	                    #sFB_MCOConveyLinxAixController210(iUDT_AixConfig := #iUDT_Configuration."210".MCO_M01,
	                                                       iv_AixInputsModule := #iUDT_MotorInput210,
	                                                       ix_24vOk := #ix_24vOk,
	                                                       ix_SimulationModeActive := "DB_Memory".Simulation,
	                                                       ii_MotorPositionId := 1,
	                                                       qUDT_HMIStatus => #iqUDT_WorkstationStatus."210".MCO_M01,
	                                                       iqv_AixOutputsModule := #iqUDT_MotorOutput210,
	                                                       iqUDT_ConveyorInterface := #sUDT_Interface210,
	                                                       iqUDT_MCOStatistics := #iqUDT_WorkstationStatistics."210".MCO_M01);
	                END_REGION
	            END_REGION

	            REGION 211

	                REGION Displacement

	                    #sFB_Displacement211(#sUDT_Interface211);

	                END_REGION

	                REGION RAT

	                    IF #iUDT_Configuration.GlobalConfig.StationVariant = 1 OR #iUDT_Configuration.GlobalConfig.StationVariant = 2 THEN
	                        #sUDT_Handshake211C := #sUDT_Handshake190;
	                    ELSIF #iUDT_Configuration.GlobalConfig.StationVariant = 3 THEN
	                        #sUDT_Handshake211D := #sUDT_Handshake590;
	                    END_IF;


	                    #sFB_RightAngledTransfer211(iUDT_Configuration := #iUDT_Configuration."211".RightAngledTransfer,
	                                                iUDT_LowerConveyorConfiguration := #iUDT_Configuration."210".Conveyor,
	                                                iUDT_UpperConveyorConfiguration := #iUDT_Configuration."211".Conveyor,
	                                                iUDT_PECConfiguration := #iUDT_Configuration."210".PEC_EoS,
	                                                ii_DestinationA := 0,
	                                                ii_DestinationB := 0,
	                                                ii_DestinationC := 2,
	                                                ii_DestinationD := 0,
	                                                ix_HardwareOk := #iUDT_HardwareOk."210",
	                                                ix_400vOk := #ix_400vOk,
	                                                ix_24vOk := #ix_24vOk,
	                                                ix_SafetyOk := #ix_SafetyOk,
	                                                ix_AirPressureOk := #ix_AirPressureOk,
	                                                ix_SectionIsDown := #ix_SectionIsDown211,
	                                                ix_SectionIsUp := #ix_SectionIsUp211,
	                                                ix_ConveyorAAuto := false,
	                                                ix_ConveyorBAuto := false,
	                                                ix_ConveyorCAuto := #iqUDT_WorkstationCommonStatus."190".AutoON,
	                                                ix_ConveyorDAuto := false,
	                                                ix_PEC := #iUDT_MotorInput210.AllSensorPortInputs.LeftSensor,
	                                                ix_ExternalReceiveRequestA := FALSE,
	                                                ix_ExternalReceiveRequestB := FALSE,
	                                                ix_ExternalReceiveRequestC := #sx_LeftPushOutActiveStation1,
	                                                ix_ExternalReceiveRequestD := FALSE,
	                                                ix_PECInfeedC := #iqUDT_WorkstationStatus."190".PEC_EoS.PEC,
	                                                qUDT_HMIRATStatus => #iqUDT_WorkstationStatus."211".RightAngledTransfer,
	                                                qUDT_HMIConveyorStatus => #iqUDT_WorkstationStatus."210".Conveyor,
	                                                qUDT_HMIPECStatus => #iqUDT_WorkstationStatus."210".PEC_EoS,
	                                                qUDT_RATStatus => #iqUDT_WorkstationCommonStatus."211",
	                                                qUDT_ConveyorStatus => #iqUDT_WorkstationCommonStatus."210",
	                                                qx_PopupControl => #qx_PopupControl211,
	                                                qx_ExternalSendRequestA => #tx_dummy,
	                                                qx_ExternalSendRequestB => #tx_dummy,
	                                                qx_ExternalSendRequestC => #tx_dummy,
	                                                qx_ExternalSendRequestD => #tx_dummy,
	                                                iqUDT_EquipmentControl := #iqUDT_EquipmentControl,
	                                                iqUDT_RATCommand := #iqUDT_WorkstationCommands."211".RightAngledTransfer,
	                                                iqUDT_ConveyorCommand := #iqUDT_WorkstationCommands."210".Conveyor,
	                                                iqUDT_RATStatistics := #iqUDT_WorkstationStatistics."211".RightAngledTransfer,
	                                                iqUDT_ConveyorStatistics := #iqUDT_WorkstationStatistics."210".Conveyor,
	                                                iqUDT_PECStatistics := #iqUDT_WorkstationStatistics."210".PEC_EoS,
	                                                iqUDT_HandShakeConveyorA := #tUDT_DummyConveyorHandshake,
	                                                iqUDT_HandShakeConveyorB := #sUDT_Handshake210,
	                                                iqUDT_HandShakeConveyorC := #sUDT_Handshake211C,
	                                                iqUDT_HandShakeConveyorD := #sUDT_Handshake211D,
	                                                iqUDT_LowerConveyorInterface := #sUDT_Interface210,
	                                                iqUDT_UpperConveyorInterface := #sUDT_Interface211,
	                                                iqUDT_RATPositioning := #iqUDT_RATPositioning210,
	                                                iqUDT_BladeStopEoSInterface := #tUDT_DummyBladeStop,
	                                                iqUDT_BladeStopBoSInterface := #tUDT_DummyBladeStop);

	                END_REGION

	                IF #iUDT_Configuration.GlobalConfig.StationVariant = 1 OR #iUDT_Configuration.GlobalConfig.StationVariant = 2 THEN
	                    #sUDT_Handshake190 := #sUDT_Handshake211C;
	                ELSIF #iUDT_Configuration.GlobalConfig.StationVariant = 3 THEN
	                    #sUDT_Handshake590 := #sUDT_Handshake211D;
	                END_IF;


	                REGION MCO

	                    #sFB_MCOConveyLinxAixController211(iUDT_AixConfig := #iUDT_Configuration."211".MCO_M01,
	                                                       iv_AixInputsModule := #iUDT_MotorInput210,
	                                                       ii_PositionSetpoint := #iqUDT_RATPositioning210.Upper.EndPosition,
	                                                       ix_24vOk := #ix_24vOk,
	                                                       ix_SimulationModeActive := "DB_Memory".Simulation,
	                                                       ii_MotorPositionId := 2,
	                                                       ix_StartPositioning := #iqUDT_RATPositioning210.Upper.Start,
	                                                       ix_ResetPosition := #iqUDT_RATPositioning210.Upper.ResetPosition,
	                                                       qUDT_HMIStatus => #iqUDT_WorkstationStatus."211".MCO_M01,
	                                                       qx_Positioned => #iqUDT_RATPositioning210.Upper.Done,
	                                                       iqv_AixOutputsModule := #iqUDT_MotorOutput210,
	                                                       iqUDT_ConveyorInterface := #sUDT_Interface211,
	                                                       iqUDT_MCOStatistics := #iqUDT_WorkstationStatistics."211".MCO_M01);
	                END_REGION

	            END_REGION

	            REGION 220

	                REGION Displacement

	                    #sFB_Displacement220(#sUDT_Interface220);

	                END_REGION

	                REGION MCO

	                    #sFB_MCOConveyLinxAixController220(iUDT_AixConfig := #iUDT_Configuration."220".MCO_M01,
	                                                       iv_AixInputsModule := #iUDT_MotorInput220,
	                                                       ii_PositionSetpoint := #iqUDT_RATPositioning220.Lower.EndPosition,
	                                                       ix_24vOk := #ix_24vOk,
	                                                       ix_SimulationModeActive := "DB_Memory".Simulation,
	                                                       ii_MotorPositionId := 1,
	                                                       ix_StartPositioning := #iqUDT_RATPositioning220.Lower.Start,
	                                                       ix_ResetPosition := #iqUDT_RATPositioning220.Lower.ResetPosition,
	                                                       qUDT_HMIStatus => #iqUDT_WorkstationStatus."220".MCO_M01,
	                                                       qx_Positioned => #iqUDT_RATPositioning220.Lower.Done,
	                                                       iqv_AixOutputsModule := #iqUDT_MotorOutput220,
	                                                       iqUDT_ConveyorInterface := #sUDT_Interface220,
	                                                       iqUDT_MCOStatistics := #iqUDT_WorkstationStatistics."220".MCO_M01);
	                END_REGION
	            END_REGION

	            REGION 221

	                REGION Displacement

	                    #sFB_Displacement221(#sUDT_Interface221);

	                END_REGION

	                REGION RAT

	                    IF #iUDT_Configuration.GlobalConfig.StationVariant = 1 OR #iUDT_Configuration.GlobalConfig.StationVariant = 2 THEN
	                        #sUDT_Handshake221C := #sUDT_Handshake350;
	                    ELSIF #iUDT_Configuration.GlobalConfig.StationVariant = 3 THEN
	                        #sUDT_Handshake221D := #sUDT_Handshake750;
	                    END_IF;


	                    #sFB_RightAngledTransfer221(iUDT_Configuration := #iUDT_Configuration."221".RightAngledTransfer,
	                                                iUDT_LowerConveyorConfiguration := #iUDT_Configuration."220".Conveyor,
	                                                iUDT_UpperConveyorConfiguration := #iUDT_Configuration."221".Conveyor,
	                                                iUDT_PECConfiguration := #iUDT_Configuration."220".PEC_EoS,
	                                                ii_DestinationA := 2,
	                                                ii_DestinationB := 0,
	                                                ii_DestinationC := 2,
	                                                ii_DestinationD := 0,
	                                                ix_HardwareOk := #iUDT_HardwareOk."220",
	                                                ix_400vOk := #ix_400vOk,
	                                                ix_24vOk := #ix_24vOk,
	                                                ix_SafetyOk := #ix_SafetyOk,
	                                                ix_AirPressureOk := #ix_AirPressureOk,
	                                                ix_SectionIsDown := #ix_SectionIsDown221,
	                                                ix_SectionIsUp := #ix_SectionIsUp221,
	                                                ix_ConveyorAAuto := #iqUDT_WorkstationCommonStatus."210".AutoON,
	                                                ix_ConveyorBAuto := false,
	                                                ix_ConveyorCAuto := #iqUDT_WorkstationCommonStatus."350".AutoON,
	                                                ix_ConveyorDAuto := false,
	                                                ix_PEC := #iUDT_MotorInput220.AllSensorPortInputs.LeftSensor,
	                                                ix_ExternalReceiveRequestA := NOT #iqUDT_WorkstationStatus."210".PEC_EoS.PEC,
	                                                ix_ExternalReceiveRequestB := FALSE,
	                                                ix_ExternalReceiveRequestC := NOT #iqUDT_WorkstationStatus."350".PEC_EoS.PEC,
	                                                ix_ExternalReceiveRequestD := TRUE,
	                                                ix_PECInfeedA := #iqUDT_WorkstationStatus."210".PEC_EoS.PEC,
	                                                ix_PECInfeedC := #iqUDT_WorkstationStatus."350".PEC_EoS.PEC,
	                                                qUDT_HMIRATStatus => #iqUDT_WorkstationStatus."221".RightAngledTransfer,
	                                                qUDT_HMIConveyorStatus => #iqUDT_WorkstationStatus."220".Conveyor,
	                                                qUDT_HMIPECStatus => #iqUDT_WorkstationStatus."220".PEC_EoS,
	                                                qUDT_RATStatus => #iqUDT_WorkstationCommonStatus."221",
	                                                qUDT_ConveyorStatus => #iqUDT_WorkstationCommonStatus."220",
	                                                qx_PopupControl => #qx_PopupControl221,
	                                                qx_ExternalSendRequestA => #tx_dummy,
	                                                qx_ExternalSendRequestB => #tx_dummy,
	                                                qx_ExternalSendRequestC => #tx_dummy,
	                                                qx_ExternalSendRequestD => #tx_dummy,
	                                                iqUDT_EquipmentControl := #iqUDT_EquipmentControl,
	                                                iqUDT_RATCommand := #iqUDT_WorkstationCommands."221".RightAngledTransfer,
	                                                iqUDT_ConveyorCommand := #iqUDT_WorkstationCommands."220".Conveyor,
	                                                iqUDT_RATStatistics := #iqUDT_WorkstationStatistics."221".RightAngledTransfer,
	                                                iqUDT_ConveyorStatistics := #iqUDT_WorkstationStatistics."220".Conveyor,
	                                                iqUDT_PECStatistics := #iqUDT_WorkstationStatistics."220".PEC_EoS,
	                                                iqUDT_HandShakeConveyorA := #sUDT_Handshake210,
	                                                iqUDT_HandShakeConveyorB := #iqUDT_HandshakeDownstream220,
	                                                iqUDT_HandShakeConveyorC := #sUDT_Handshake221C,
	                                                iqUDT_HandShakeConveyorD := #sUDT_Handshake221D,
	                                                iqUDT_LowerConveyorInterface := #sUDT_Interface220,
	                                                iqUDT_UpperConveyorInterface := #sUDT_Interface221,
	                                                iqUDT_RATPositioning := #iqUDT_RATPositioning220,
	                                                iqUDT_BladeStopEoSInterface := #tUDT_DummyBladeStop,
	                                                iqUDT_BladeStopBoSInterface := #tUDT_DummyBladeStop);

	                END_REGION

	                IF #iUDT_Configuration.GlobalConfig.StationVariant = 1 OR #iUDT_Configuration.GlobalConfig.StationVariant = 2 THEN
	                    #sUDT_Handshake350 := #sUDT_Handshake221C;
	                ELSIF #iUDT_Configuration.GlobalConfig.StationVariant = 3 THEN
	                    #sUDT_Handshake750 := #sUDT_Handshake221D;
	                END_IF;

	                REGION MCO

	                    #sFB_MCOConveyLinxAixController221(iUDT_AixConfig := #iUDT_Configuration."221".MCO_M01,
	                                                       iv_AixInputsModule := #iUDT_MotorInput220,
	                                                       ii_PositionSetpoint := #iqUDT_RATPositioning220.Upper.EndPosition,
	                                                       ix_24vOk := #ix_24vOk,
	                                                       ix_SimulationModeActive := "DB_Memory".Simulation,
	                                                       ii_MotorPositionId := 2,
	                                                       ix_StartPositioning := #iqUDT_RATPositioning220.Upper.Start,
	                                                       ix_ResetPosition := #iqUDT_RATPositioning220.Upper.ResetPosition,
	                                                       qUDT_HMIStatus => #iqUDT_WorkstationStatus."221".MCO_M01,
	                                                       qx_Positioned => #iqUDT_RATPositioning220.Upper.Done,
	                                                       iqv_AixOutputsModule := #iqUDT_MotorOutput220,
	                                                       iqUDT_ConveyorInterface := #sUDT_Interface221,
	                                                       iqUDT_MCOStatistics := #iqUDT_WorkstationStatistics."221".MCO_M01);
	                END_REGION
	            END_REGION

	            REGION 310

	                REGION Displacement

	                    #sFB_Displacement310(#sUDT_Interface310);

	                END_REGION

	                REGION EOS
	                    #sFB_PEC310(ix_PEC := NOT #iUDT_MotorInput310.AllSensorPortInputs.LeftSensor,
	                                iUDT_PECConfiguration := #iUDT_Configuration."310".PEC_Eos,
	                                qx_PECFiltered => #tx_dummy,
	                                qUDT_HMIStatus => #iqUDT_WorkstationStatus."310".PEC_EoS,
	                                iqUDT_ConveyorInterface := #sUDT_Interface310,
	                                iqUDT_PECStatistics := #iqUDT_WorkstationStatistics."310".PEC_EoS);

	                END_REGION

	                REGION Conveyor

	                    #sFB_Conveyor310(iUDT_ConveyorConfiguration := #iUDT_Configuration."310".Conveyor,
	                                     idi_PECEoSDistance := #iUDT_Configuration."310".PEC_Eos.Distance,
	                                     idi_PECBoSDistance := 0,
	                                     ii_ExternalSpeed := 0,
	                                     ix_SafetyOk := #ix_SafetyOk,
	                                     ix_24vOk := #ix_24vOk,
	                                     ix_400vOk := #ix_400vOk,
	                                     ix_HardwareOk := #iUDT_HardwareOk."310",
	                                     ix_PECEoS := #iqUDT_WorkstationStatus."310".PEC_EoS.PEC,
	                                     ix_PECBoS := TRUE,
	                                     ix_ReverseDirection := FALSE,
	                                     ix_ExternalRequestDieBack := FALSE,
	                                     ix_ExternalRequestHold := #sx_LeftExternalRequestHold310,
	                                     ix_ResetEnergySave := FALSE,
	                                     qUDT_HMIStatus => #iqUDT_WorkstationStatus."310".Conveyor,
	                                     qUDT_Status => #iqUDT_WorkstationCommonStatus."310",
	                                     iqUDT_EquipmentControl := #iqUDT_EquipmentControl,
	                                     iqUDT_ConveyorCommand := #iqUDT_WorkstationCommands."310".Conveyor,
	                                     iqUDT_ConveyorInterface := #sUDT_Interface310,
	                                     iqUDT_HandShakeUp := #tUDT_DummyConveyorHandshake,
	                                     iqUDT_HandShake := #sUDT_Handshake310,
	                                     iqUDT_Statistics := #iqUDT_WorkstationStatistics."310".Conveyor);
	                END_REGION

	                REGION MCO

	                    #sFB_MCOConveyLinxAixController310(iUDT_AixConfig := #iUDT_Configuration."310".MCO_M01,
	                                                       iv_AixInputsModule := #iUDT_MotorInput310,
	                                                       ix_24vOk := #ix_24vOk,
	                                                       ix_SimulationModeActive := "DB_Memory".Simulation,
	                                                       ii_MotorPositionId := 1,
	                                                       qUDT_HMIStatus => #iqUDT_WorkstationStatus."310".MCO_M01,
	                                                       iqv_AixOutputsModule := #iqUDT_MotorOutput310,
	                                                       iqUDT_ConveyorInterface := #sUDT_Interface310,
	                                                       iqUDT_MCOStatistics := #iqUDT_WorkstationStatistics."310".MCO_M01);
	                END_REGION

	            END_REGION

	            REGION 320

	                REGION Displacement

	                    #sFB_Displacement320(#sUDT_Interface320);

	                END_REGION

	                REGION EOS
	                    #sFB_PEC320(ix_PEC := NOT #iUDT_MotorInput310.AllSensorPortInputs.RightSensor,
	                                iUDT_PECConfiguration := #iUDT_Configuration."320".PEC_Eos,
	                                qx_PECFiltered => #tx_dummy,
	                                qUDT_HMIStatus => #iqUDT_WorkstationStatus."320".PEC_EoS,
	                                iqUDT_ConveyorInterface := #sUDT_Interface320,
	                                iqUDT_PECStatistics := #iqUDT_WorkstationStatistics."320".PEC_EoS);


	                END_REGION

	                REGION Conveyor

	                    #sFB_Conveyor320(iUDT_ConveyorConfiguration := #iUDT_Configuration."320".Conveyor,
	                                     idi_PECEoSDistance := #iUDT_Configuration."320".PEC_Eos.Distance,
	                                     idi_PECBoSDistance := 0,
	                                     ii_ExternalSpeed := 0,
	                                     ix_SafetyOk := #ix_SafetyOk,
	                                     ix_24vOk := #ix_24vOk,
	                                     ix_400vOk := #ix_400vOk,
	                                     ix_HardwareOk := #iUDT_HardwareOk."320",
	                                     ix_PECEoS := #iqUDT_WorkstationStatus."320".PEC_EoS.PEC,
	                                     ix_PECBoS := TRUE,
	                                     ix_ReverseDirection := FALSE,
	                                     ix_ExternalRequestDieBack := FALSE,
	                                     ix_ExternalRequestHold := #sx_LeftExternalRequestHold320,
	                                     ix_ResetEnergySave := FALSE,
	                                     qUDT_HMIStatus => #iqUDT_WorkstationStatus."320".Conveyor,
	                                     qUDT_Status => #iqUDT_WorkstationCommonStatus."320",
	                                     iqUDT_EquipmentControl := #iqUDT_EquipmentControl,
	                                     iqUDT_ConveyorCommand := #iqUDT_WorkstationCommands."320".Conveyor,
	                                     iqUDT_ConveyorInterface := #sUDT_Interface320,
	                                     iqUDT_HandShakeUp := #sUDT_Handshake310,
	                                     iqUDT_HandShake := #sUDT_Handshake320,
	                                     iqUDT_Statistics := #iqUDT_WorkstationStatistics."320".Conveyor);
	                END_REGION

	                REGION MCO

	                    #sFB_MCOConveyLinxAixController320(iUDT_AixConfig := #iUDT_Configuration."320".MCO_M01,
	                                                       iv_AixInputsModule := #iUDT_MotorInput310,
	                                                       ix_24vOk := #ix_24vOk,
	                                                       ix_SimulationModeActive := "DB_Memory".Simulation,
	                                                       ii_MotorPositionId := 2,
	                                                       qUDT_HMIStatus => #iqUDT_WorkstationStatus."320".MCO_M01,
	                                                       iqv_AixOutputsModule := #iqUDT_MotorOutput310,
	                                                       iqUDT_ConveyorInterface := #sUDT_Interface320,
	                                                       iqUDT_MCOStatistics := #iqUDT_WorkstationStatistics."320".MCO_M01);
	                END_REGION

	            END_REGION

	            REGION 330

	                REGION Displacement

	                    #sFB_Displacement330(#sUDT_Interface330);

	                END_REGION

	                REGION EOS
	                    #sFB_PEC330(ix_PEC := NOT #iUDT_MotorInput330.AllSensorPortInputs.LeftSensor,
	                                iUDT_PECConfiguration := #iUDT_Configuration."330".PEC_Eos,
	                                qx_PECFiltered => #tx_dummy,
	                                qUDT_HMIStatus => #iqUDT_WorkstationStatus."330".PEC_EoS,
	                                iqUDT_ConveyorInterface := #sUDT_Interface330,
	                                iqUDT_PECStatistics := #iqUDT_WorkstationStatistics."330".PEC_EoS);


	                END_REGION

	                REGION Conveyor

	                    #sFB_Conveyor330(iUDT_ConveyorConfiguration := #iUDT_Configuration."330".Conveyor,
	                                     idi_PECEoSDistance := #iUDT_Configuration."330".PEC_Eos.Distance,
	                                     idi_PECBoSDistance := 0,
	                                     ii_ExternalSpeed := 0,
	                                     ix_SafetyOk := #ix_SafetyOk,
	                                     ix_24vOk := #ix_24vOk,
	                                     ix_400vOk := #ix_400vOk,
	                                     ix_HardwareOk := #iUDT_HardwareOk."330",
	                                     ix_PECEoS := #iqUDT_WorkstationStatus."330".PEC_EoS.PEC,
	                                     ix_PECBoS := TRUE,
	                                     ix_ReverseDirection := FALSE,
	                                     ix_ExternalRequestDieBack := FALSE,
	                                     ix_ExternalRequestHold := #sx_LeftExternalRequestHold330,
	                                     ix_ResetEnergySave := FALSE,
	                                     qUDT_HMIStatus => #iqUDT_WorkstationStatus."330".Conveyor,
	                                     qUDT_Status => #iqUDT_WorkstationCommonStatus."330",
	                                     iqUDT_EquipmentControl := #iqUDT_EquipmentControl,
	                                     iqUDT_ConveyorCommand := #iqUDT_WorkstationCommands."330".Conveyor,
	                                     iqUDT_ConveyorInterface := #sUDT_Interface330,
	                                     iqUDT_HandShakeUp := #sUDT_Handshake320,
	                                     iqUDT_HandShake := #sUDT_Handshake330,
	                                     iqUDT_Statistics := #iqUDT_WorkstationStatistics."330".Conveyor);
	                END_REGION

	                REGION MCO

	                    #sFB_MCOConveyLinxAixController330(iUDT_AixConfig := #iUDT_Configuration."330".MCO_M01,
	                                                       iv_AixInputsModule := #iUDT_MotorInput330,
	                                                       ix_24vOk := #ix_24vOk,
	                                                       ix_SimulationModeActive := "DB_Memory".Simulation,
	                                                       ii_MotorPositionId := 1,
	                                                       qUDT_HMIStatus => #iqUDT_WorkstationStatus."330".MCO_M01,
	                                                       iqv_AixOutputsModule := #iqUDT_MotorOutput330,
	                                                       iqUDT_ConveyorInterface := #sUDT_Interface330,
	                                                       iqUDT_MCOStatistics := #iqUDT_WorkstationStatistics."330".MCO_M01);
	                END_REGION
	            END_REGION

	            REGION 340

	                REGION Displacement

	                    #sFB_Displacement340(#sUDT_Interface340);

	                END_REGION

	                REGION EOS
	                    #sFB_PEC340(ix_PEC := NOT #iUDT_MotorInput330.AllSensorPortInputs.RightSensor,
	                                iUDT_PECConfiguration := #iUDT_Configuration."340".PEC_Eos,
	                                qx_PECFiltered => #tx_dummy,
	                                qUDT_HMIStatus => #iqUDT_WorkstationStatus."340".PEC_EoS,
	                                iqUDT_ConveyorInterface := #sUDT_Interface340,
	                                iqUDT_PECStatistics := #iqUDT_WorkstationStatistics."340".PEC_EoS);


	                END_REGION


	                REGION Conveyor

	                    #sFB_Conveyor340(iUDT_ConveyorConfiguration := #iUDT_Configuration."340".Conveyor,
	                                     idi_PECEoSDistance := #iUDT_Configuration."340".PEC_Eos.Distance,
	                                     idi_PECBoSDistance := 0,
	                                     ii_ExternalSpeed := 0,
	                                     ix_SafetyOk := #ix_SafetyOk,
	                                     ix_24vOk := #ix_24vOk,
	                                     ix_400vOk := #ix_400vOk,
	                                     ix_HardwareOk := #iUDT_HardwareOk."340",
	                                     ix_PECEoS := #iqUDT_WorkstationStatus."340".PEC_EoS.PEC,
	                                     ix_PECBoS := TRUE,
	                                     ix_ReverseDirection := FALSE,
	                                     ix_ExternalRequestDieBack := FALSE,
	                                     ix_ExternalRequestHold := #sx_LeftExternalRequestHold340,
	                                     ix_ResetEnergySave := FALSE,
	                                     qUDT_HMIStatus => #iqUDT_WorkstationStatus."340".Conveyor,
	                                     qUDT_Status => #iqUDT_WorkstationCommonStatus."340",
	                                     iqUDT_EquipmentControl := #iqUDT_EquipmentControl,
	                                     iqUDT_ConveyorCommand := #iqUDT_WorkstationCommands."340".Conveyor,
	                                     iqUDT_ConveyorInterface := #sUDT_Interface340,
	                                     iqUDT_HandShakeUp := #sUDT_Handshake330,
	                                     iqUDT_HandShake := #sUDT_Handshake340,
	                                     iqUDT_Statistics := #iqUDT_WorkstationStatistics."340".Conveyor);
	                END_REGION

	                REGION MCO

	                    #sFB_MCOConveyLinxAixController340(iUDT_AixConfig := #iUDT_Configuration."340".MCO_M01,
	                                                       iv_AixInputsModule := #iUDT_MotorInput330,
	                                                       ix_24vOk := #ix_24vOk,
	                                                       ix_SimulationModeActive := "DB_Memory".Simulation,
	                                                       ii_MotorPositionId := 2,
	                                                       qUDT_HMIStatus => #iqUDT_WorkstationStatus."340".MCO_M01,
	                                                       iqv_AixOutputsModule := #iqUDT_MotorOutput330,
	                                                       iqUDT_ConveyorInterface := #sUDT_Interface340,
	                                                       iqUDT_MCOStatistics := #iqUDT_WorkstationStatistics."340".MCO_M01);
	                END_REGION
	            END_REGION

	            REGION 350

	                REGION Displacement

	                    #sFB_Displacement350(#sUDT_Interface350);

	                END_REGION

	                REGION EOS
	                    #sFB_PEC350(ix_PEC := NOT #iUDT_MotorInput350.AllSensorPortInputs.LeftSensor,
	                                iUDT_PECConfiguration := #iUDT_Configuration."350".PEC_Eos,
	                                qx_PECFiltered => #tx_dummy,
	                                qUDT_HMIStatus => #iqUDT_WorkstationStatus."350".PEC_EoS,
	                                iqUDT_ConveyorInterface := #sUDT_Interface350,
	                                iqUDT_PECStatistics := #iqUDT_WorkstationStatistics."350".PEC_EoS);

	                END_REGION

	                REGION Conveyor

	                    #sUDT_Handshake350.RTR := #sUDT_Handshake350.RTR OR #iqUDT_WorkstationStatus."350".PEC_EoS.PEC;

	                    #sFB_Conveyor350(iUDT_ConveyorConfiguration := #iUDT_Configuration."350".Conveyor,
	                                     idi_PECEoSDistance := #iUDT_Configuration."350".PEC_Eos.Distance,
	                                     idi_PECBoSDistance := 0,
	                                     ii_ExternalSpeed := 0,
	                                     ix_SafetyOk := #ix_SafetyOk,
	                                     ix_24vOk := #ix_24vOk,
	                                     ix_400vOk := #ix_400vOk,
	                                     ix_HardwareOk := #iUDT_HardwareOk."350",
	                                     ix_PECEoS := #iqUDT_WorkstationStatus."350".PEC_EoS.PEC,
	                                     ix_PECBoS := TRUE,
	                                     ix_ReverseDirection := FALSE,
	                                     ix_ExternalRequestDieBack := FALSE,
	                                     ix_ExternalRequestHold := #sx_LeftExternalRequestHold350,
	                                     ix_ResetEnergySave := FALSE,
	                                     qUDT_HMIStatus => #iqUDT_WorkstationStatus."350".Conveyor,
	                                     qUDT_Status => #iqUDT_WorkstationCommonStatus."350",
	                                     iqUDT_EquipmentControl := #iqUDT_EquipmentControl,
	                                     iqUDT_ConveyorCommand := #iqUDT_WorkstationCommands."350".Conveyor,
	                                     iqUDT_ConveyorInterface := #sUDT_Interface350,
	                                     iqUDT_HandShakeUp := #sUDT_Handshake340,
	                                     iqUDT_HandShake := #sUDT_Handshake350,
	                                     iqUDT_Statistics := #iqUDT_WorkstationStatistics."350".Conveyor);
	                END_REGION

	                REGION MCO

	                    #sFB_MCOConveyLinxAixController350(iUDT_AixConfig := #iUDT_Configuration."350".MCO_M01,
	                                                       iv_AixInputsModule := #iUDT_MotorInput350,
	                                                       ix_24vOk := #ix_24vOk,
	                                                       ix_SimulationModeActive := "DB_Memory".Simulation,
	                                                       ii_MotorPositionId := 1,
	                                                       qUDT_HMIStatus => #iqUDT_WorkstationStatus."350".MCO_M01,
	                                                       iqv_AixOutputsModule := #iqUDT_MotorOutput350,
	                                                       iqUDT_ConveyorInterface := #sUDT_Interface350,
	                                                       iqUDT_MCOStatistics := #iqUDT_WorkstationStatistics."350".MCO_M01);
	                END_REGION
	            END_REGION

	            REGION 360

	                REGION Displacement
	                    #sFB_Displacement360(#sUDT_Interface360);

	                END_REGION


	                REGION Conveyor

	                    #sUDT_Handshake360.RTR := TRUE;

	                    #sFB_Conveyor360(iUDT_ConveyorConfiguration := #iUDT_Configuration."360".Conveyor,
	                                     idi_PECEoSDistance := 0,
	                                     idi_PECBoSDistance := 0,
	                                     ii_ExternalSpeed := 0,
	                                     ix_SafetyOk := #ix_SafetyOk,
	                                     ix_24vOk := #ix_24vOk,
	                                     ix_400vOk := #ix_400vOk,
	                                     ix_HardwareOk := #iUDT_HardwareOk."360",
	                                     ix_PECEoS := TRUE,
	                                     ix_PECBoS := TRUE,
	                                     ix_ReverseDirection := false,
	                                     ix_ExternalRequestDieBack := false,
	                                     ix_ExternalRequestHold := #sx_Hold360,
	                                     ix_ResetEnergySave := false,
	                                     qUDT_HMIStatus => #iqUDT_WorkstationStatus."360".Conveyor,
	                                     qUDT_Status => #iqUDT_WorkstationCommonStatus."360",
	                                     iqUDT_EquipmentControl := #iqUDT_EquipmentControl,
	                                     iqUDT_ConveyorCommand := #iqUDT_WorkstationCommands."360".Conveyor,
	                                     iqUDT_ConveyorInterface := #sUDT_Interface360,
	                                     iqUDT_HandShakeUp := #sUDT_HandshakeUp360,
	                                     iqUDT_HandShake := #sUDT_Handshake360,
	                                     iqUDT_Statistics := #iqUDT_WorkstationStatistics."360".Conveyor);

	                END_REGION


	                REGION MCO
	                    #sFB_MCOConveyLinxAixController360(iUDT_AixConfig := #iUDT_Configuration."360".MCO_M01,
	                                                       iv_AixInputsModule := #iUDT_MotorInput360,
	                                                       ii_MotorPositionId := 1,
	                                                       ix_24vOk := #ix_24vOk,
	                                                       ix_SimulationModeActive := "DB_Memory".Simulation,
	                                                       qUDT_HMIStatus => #iqUDT_WorkstationStatus."360".MCO_M01,
	                                                       iqv_AixOutputsModule := #iqUDT_MotorOutput360,
	                                                       iqUDT_ConveyorInterface := #sUDT_Interface360,
	                                                       iqUDT_MCOStatistics := #iqUDT_WorkstationStatistics."360".MCO_M01);

	                END_REGION

	            END_REGION

	            REGION 370
	                REGION Displacement
	                    #sFB_Displacement370(#sUDT_Interface370);

	                END_REGION

	                REGION Conveyor

	                    #sUDT_Handshake370.RTR := TRUE;

	                    #sFB_Conveyor370(iUDT_ConveyorConfiguration := #iUDT_Configuration."370".Conveyor,
	                                     idi_PECEoSDistance := 0,
	                                     idi_PECBoSDistance := 0,
	                                     ii_ExternalSpeed := 0,
	                                     ix_SafetyOk := #ix_SafetyOk,
	                                     ix_24vOk := #ix_24vOk,
	                                     ix_400vOk := #ix_400vOk,
	                                     ix_HardwareOk := #iUDT_HardwareOk."360",
	                                     ix_PECEoS := TRUE,
	                                     ix_PECBoS := TRUE,
	                                     ix_ReverseDirection := false,
	                                     ix_ExternalRequestDieBack := false,
	                                     ix_ExternalRequestHold := #sx_Hold370,
	                                     ix_ResetEnergySave := false,
	                                     qUDT_HMIStatus => #iqUDT_WorkstationStatus."370".Conveyor,
	                                     qUDT_Status => #iqUDT_WorkstationCommonStatus."370",
	                                     iqUDT_EquipmentControl := #iqUDT_EquipmentControl,
	                                     iqUDT_ConveyorCommand := #iqUDT_WorkstationCommands."370".Conveyor,
	                                     iqUDT_ConveyorInterface := #sUDT_Interface370,
	                                     iqUDT_HandShakeUp := #sUDT_HandshakeUp370,
	                                     iqUDT_HandShake := #sUDT_Handshake370,
	                                     iqUDT_Statistics := #iqUDT_WorkstationStatistics."370".Conveyor);

	                END_REGION


	                REGION MCO
	                    #sFB_MCOConveyLinxAixController370(iUDT_AixConfig := #iUDT_Configuration."370".MCO_M01,
	                                                       iv_AixInputsModule := #iUDT_MotorInput360,
	                                                       ii_MotorPositionId := 2,
	                                                       ii_PositionSetpoint := 0,
	                                                       ix_24vOk := #ix_24vOk,
	                                                       ix_SimulationModeActive := "DB_Memory".Simulation,
	                                                       ix_StartPositioning := false,
	                                                       ix_ResetPosition := false,
	                                                       qUDT_HMIStatus => #iqUDT_WorkstationStatus."370".MCO_M01,
	                                                       iqv_AixOutputsModule := #iqUDT_MotorOutput360,
	                                                       iqUDT_ConveyorInterface := #sUDT_Interface370,
	                                                       iqUDT_MCOStatistics := #iqUDT_WorkstationStatistics."370".MCO_M01);
	                END_REGION

	            END_REGION

	        END_REGION
	    END_IF;

	END_REGION

	REGION 6 - Right station

	    IF #iUDT_Configuration.GlobalConfig.StationVariant = 1 OR #iUDT_Configuration.GlobalConfig.StationVariant = 3 THEN

	        REGION 6.1 - Indexing

	            // Start indexing after request if there are empty stations and no pushout is active
	            IF #sx_RightActivateIndex AND #si_RightEmptyStations > 0
	                AND NOT (#sx_RightPushOutActiveStation1
	                OR #sx_RightPushOutActiveStation2
	                OR #sx_RightPushOutActiveStation3
	                OR #sx_RightPushOutActiveStation4
	                OR #sx_RightPushOutActiveStation5)
	            THEN

	                #sx_RightIndexing := TRUE;

	            END_IF;


	            IF NOT #sx_RightIndexing THEN                                      // If there is no indexing in progress

	                #si_RightDestinationD541 := 0;                                // Reset RAT destination
	                #sx_RightExternalRequestHold550 := TRUE;                      // Hold station conveyors
	                #sx_RightExternalRequestHold560 := TRUE;
	                #sx_RightExternalRequestHold570 := TRUE;
	                #sx_RightExternalRequestHold580 := TRUE;
	                #sx_RightExternalRequestHold590 := TRUE;

	            ELSE

	                IF #sR_TRIG_PEC540.Q AND #si_RightEmptyStations > 0 THEN       //Count down empty stations after diverting a tote into station
	                    #si_RightEmptyStations -= 1;
	                END_IF;

	                #si_RightDestinationD541 := 4;                               // Set RAT destination
	                #sx_RightExternalRequestHold550 := FALSE;                    // Release hold of station conveyors
	                #sx_RightExternalRequestHold560 := FALSE;
	                #sx_RightExternalRequestHold570 := FALSE;
	                #sx_RightExternalRequestHold580 := FALSE;
	                #sx_RightExternalRequestHold590 := FALSE;

	                IF                                                           //End indexing when all totes are on position
	                    NOT #iqUDT_WorkstationStatus."550".PEC_EoS.PEC
	                    AND NOT #iqUDT_WorkstationStatus."560".PEC_EoS.PEC
	                    AND NOT #iqUDT_WorkstationStatus."570".PEC_EoS.PEC
	                    AND NOT #iqUDT_WorkstationStatus."580".PEC_EoS.PEC
	                    AND NOT #iqUDT_WorkstationStatus."590".PEC_EoS.PEC
	                    AND NOT (#sUDT_Interface550.ActualSpeed > 0) THEN

	                    #sx_RightIndexing := FALSE;

	                END_IF;
	            END_IF;

	        END_REGION

	        REGION 6.2 - Push Out

	            IF #iUDT_Configuration.GlobalConfig.RightCubbyNumbering = 1 THEN
	                #sa_RightCubby[1] := 10;
	                #sa_RightCubby[2] := 9;
	                #sa_RightCubby[3] := 8;
	                #sa_RightCubby[4] := 7;
	                #sa_RightCubby[5] := 6;
	            ELSIF #iUDT_Configuration.GlobalConfig.RightCubbyNumbering = 2 THEN
	                #sa_RightCubby[1] := 5;
	                #sa_RightCubby[2] := 4;
	                #sa_RightCubby[3] := 3;
	                #sa_RightCubby[4] := 2;
	                #sa_RightCubby[5] := 1;
	            END_IF;


	            REGION 6.2.0 - Pushout conveyors hold
	                IF #sFB_TimerOnOffDelay_Hold710.qx_DelayedSignal THEN
	                    #sx_RightExternalRequestHold710 := TRUE;
	                END_IF;

	                IF #sFB_TimerOnOffDelay_Hold720.qx_DelayedSignal THEN
	                    #sx_RightExternalRequestHold720 := TRUE;
	                END_IF;

	                IF #sFB_TimerOnOffDelay_Hold730.qx_DelayedSignal THEN
	                    #sx_RightExternalRequestHold730 := TRUE;
	                END_IF;

	                IF #sFB_TimerOnOffDelay_Hold740.qx_DelayedSignal THEN
	                    #sx_RightExternalRequestHold740 := TRUE;
	                END_IF;

	                IF #sFB_TimerOnOffDelay_Hold750.qx_DelayedSignal THEN
	                    #sx_RightExternalRequestHold750 := TRUE;
	                END_IF;
	            END_REGION

	            REGION 6.2.1 - Push Out Station 1

	                // Start automatic pushout after request if there is no indexing procedure and a tote is present on first station
	                IF #iqUDT_RightWESInterface.Field[#sa_RightCubby[1]].WES2PLC.RemoveContainer AND NOT #sx_RightIndexing
	                    AND NOT #iqUDT_WorkstationStatus."590".PEC_EoS.PEC THEN

	                    #sx_RightPushOutActiveStation1 := TRUE;
	                    #iqUDT_RightWESInterface.Field[#sa_RightCubby[1]].WES2PLC.RemoveContainer := FALSE;
	                END_IF;

	                IF #sx_RightPushOutActiveStation1 THEN                         //release hold
	                    #sx_RightExternalRequestHold590 := FALSE;

	                    IF #sFB_RightAngledTransfer611.qx_ExternalSendRequestB                   //after tote is already on RAT, hold the conveyor and end pushout procedure
	                        AND #iUDT_Configuration.GlobalConfig.StationVariant <> 3             // and station has not only right station
	                    THEN
	                        #sx_RightExternalRequestHold590 := TRUE;
	                        #sx_RightPushOutActiveStation1 := FALSE;
	                    END_IF;

	                    IF #sFB_RightAngledTransfer211.qx_ExternalSendRequestB                   //after tote is already on RAT, hold the conveyor and end pushout procedure
	                        AND #iUDT_Configuration.GlobalConfig.StationVariant = 3             // and station has only right station
	                    THEN
	                        #sx_RightExternalRequestHold590 := TRUE;
	                        #sx_RightPushOutActiveStation1 := FALSE;
	                    END_IF;

	                END_IF;

	            END_REGION

	            REGION 6.2.2 - Push Out station 2

	                IF #iqUDT_RightWESInterface.Field[#sa_RightCubby[2]].WES2PLC.RemoveContainer THEN        //set pushout to active after request
	                    #sx_RightPushOutActiveStation2 := TRUE;
	                    #iqUDT_RightWESInterface.Field[#sa_RightCubby[2]].WES2PLC.RemoveContainer := FALSE;
	                END_IF;

	                IF #sx_RightPushOutActiveStation2                               // After station is empty and tote has been detected on pushout conveyor release holds
	                    AND #iqUDT_WorkstationStatus."580".PEC_EoS.PEC
	                    AND #sFB_TimerOnOffDelay_Detect740.qx_DelayedSignal THEN

	                    #sx_RightExternalRequestHold740 := FALSE;
	                    #sx_RightExternalRequestHold750 := FALSE;

	                    FILL_BLK(IN := 0,                                             //clear tracking
	                             COUNT := REAL_TO_ULINT(DINT_TO_REAL(#iUDT_Configuration."580".Conveyor.Common.Length) * #cr_ClearTrackingModifier),
	                             OUT => #sa_TrackingArray580[0]);

	                    #sx_RightPushOutActiveStation2 := FALSE;                       //end pushout procedure

	                END_IF;


	            END_REGION

	            REGION 6.2.3 - Push Out station 3

	                IF #iqUDT_RightWESInterface.Field[#sa_RightCubby[3]].WES2PLC.RemoveContainer THEN          //set pushout to active after request
	                    #sx_RightPushOutActiveStation3 := TRUE;
	                    #iqUDT_RightWESInterface.Field[#sa_RightCubby[3]].WES2PLC.RemoveContainer := FALSE;
	                END_IF;

	                IF #sx_RightPushOutActiveStation3
	                    AND #iqUDT_WorkstationStatus."570".PEC_EoS.PEC
	                    AND #sFB_TimerOnOffDelay_Detect730.qx_DelayedSignal THEN                // After station is empty and tote has been detected on pushout conveyor release holds

	                    #sx_RightExternalRequestHold730 := FALSE;
	                    #sx_RightExternalRequestHold740 := FALSE;
	                    #sx_RightExternalRequestHold750 := FALSE;

	                    FILL_BLK(IN := 0,                                                         //clear tracking
	                             COUNT := REAL_TO_ULINT(DINT_TO_REAL(#iUDT_Configuration."570".Conveyor.Common.Length) * #cr_ClearTrackingModifier),
	                             OUT => #sa_TrackingArray570[0]);

	                    #sx_RightPushOutActiveStation3 := FALSE;                              //end pushout procedure

	                END_IF;
	            END_REGION

	            REGION 6.2.4 - Push Out station 4

	                IF #iqUDT_RightWESInterface.Field[#sa_RightCubby[4]].WES2PLC.RemoveContainer THEN              //set pushout to active after request
	                    #sx_RightPushOutActiveStation4 := TRUE;
	                    #iqUDT_RightWESInterface.Field[#sa_RightCubby[4]].WES2PLC.RemoveContainer := FALSE;
	                END_IF;

	                IF #sx_RightPushOutActiveStation4
	                    AND #iqUDT_WorkstationStatus."560".PEC_EoS.PEC
	                    AND #sFB_TimerOnOffDelay_Detect720.qx_DelayedSignal THEN                // After station is empty and tote has been detected on pushout conveyor release holds

	                    #sx_RightExternalRequestHold720 := FALSE;
	                    #sx_RightExternalRequestHold730 := FALSE;
	                    #sx_RightExternalRequestHold740 := FALSE;
	                    #sx_RightExternalRequestHold750 := FALSE;

	                    FILL_BLK(IN := 0,                                                      //clear tracking
	                             COUNT := REAL_TO_ULINT(DINT_TO_REAL(#iUDT_Configuration."560".Conveyor.Common.Length) * #cr_ClearTrackingModifier),
	                             OUT => #sa_TrackingArray560[0]);

	                    #sx_RightPushOutActiveStation4 := FALSE;                          //end pushout procedure

	                END_IF;

	            END_REGION

	            REGION 6.2.5 - Push Out station 5

	                IF #iqUDT_RightWESInterface.Field[#sa_RightCubby[5]].WES2PLC.RemoveContainer THEN          //set pushout to active after request
	                    #sx_RightPushOutActiveStation5 := TRUE;
	                    #iqUDT_RightWESInterface.Field[#sa_RightCubby[5]].WES2PLC.RemoveContainer := FALSE;
	                END_IF;

	                IF #sx_RightPushOutActiveStation5
	                    AND #iqUDT_WorkstationStatus."550".PEC_EoS.PEC
	                    AND #sFB_TimerOnOffDelay_Detect710.qx_DelayedSignal THEN                // After station is empty and tote has been detected on pushout conveyor release holds

	                    #sx_RightExternalRequestHold710 := FALSE;
	                    #sx_RightExternalRequestHold720 := FALSE;
	                    #sx_RightExternalRequestHold730 := FALSE;
	                    #sx_RightExternalRequestHold740 := FALSE;
	                    #sx_RightExternalRequestHold750 := FALSE;

	                    FILL_BLK(IN := 0,                                            //clear tracking
	                             COUNT := REAL_TO_ULINT(DINT_TO_REAL(#iUDT_Configuration."550".Conveyor.Common.Length) * #cr_ClearTrackingModifier),
	                             OUT => #sa_TrackingArray550[0]);

	                    #sx_RightPushOutActiveStation5 := FALSE;                      //end pushout procedure
	                END_IF;

	            END_REGION

	            REGION 6.2.6 - Pushout support logic

	                IF #iUDT_Configuration.GlobalConfig.PushoutsPresent AND
	                    ((#iUDT_Configuration.GlobalConfig.StationVariant = 1 OR
	                    #iUDT_Configuration.GlobalConfig.StationVariant = 3)) THEN

	                    IF (NOT #iqUDT_WorkstationStatus."550".PEC_EoS.PEC AND #sx_RightPushOutActiveStation5) OR
	                        (NOT #iqUDT_WorkstationStatus."560".PEC_EoS.PEC AND #sx_RightPushOutActiveStation4) THEN
	                        #sx_Hold760 := FALSE;

	                    ELSIF NOT (#sx_LeftPushOutActiveStation5 OR #sx_LeftPushOutActiveStation4) THEN
	                        #sx_Hold760 := TRUE; //Hold pushout conveyors
	                    END_IF;

	                    //Package present on the right side pecs, pushouts run
	                    IF (NOT #iqUDT_WorkstationStatus."570".PEC_EoS.PEC AND #sx_RightPushOutActiveStation3) OR
	                        (NOT #iqUDT_WorkstationStatus."580".PEC_EoS.PEC AND #sx_RightPushOutActiveStation2) THEN
	                        #sx_Hold770 := FALSE;

	                    ELSIF NOT (#sx_LeftPushOutActiveStation3 OR #sx_LeftPushOutActiveStation2) THEN
	                        #sx_Hold770 := TRUE; //Hold pushout conveyors
	                    END_IF;
	                END_IF;

	            END_REGION
	        END_REGION

	        REGION 6.3 WES Communication

	            REGION 6.3.1 Barcode to WES
	                IF NOT #sx_RightIndexing
	                THEN

	                    REGION 590
	                        // first position
	                        //
	                        IF NOT #sx_RightPushOutActiveStation1
	                            AND NOT #iqUDT_WorkstationStatus."590".PEC_EoS.PEC
	                            AND #sa_TrackingArray590[(#iUDT_Configuration."590".PEC_Eos.Distance / 10) - 1] > 0
	                        THEN

	                            IF #iqUDT_RightWESInterface.Field[#sa_RightCubby[1]].WES2PLC.SetContainerID THEN

	                                "DB_GIN".GIN[#sa_TrackingArray590[(#iUDT_Configuration."590".PEC_Eos.Distance / 10) - 1]].General.Identification.Barcode := #iqUDT_RightWESInterface.Field[#sa_RightCubby[1]].WES2PLC.ContainerID;
	                                #iqUDT_RightWESInterface.Field[#sa_RightCubby[1]].WES2PLC.SetContainerID := FALSE;

	                            END_IF;

	                            IF #iqUDT_RightWESInterface.Field[#sa_RightCubby[1]].PLC2WES.ContainerID <> "DB_GIN".GIN[#sa_TrackingArray590[(#iUDT_Configuration."590".PEC_Eos.Distance / 10) - 1]].General.Identification.Barcode
	                            THEN

	                                #iqUDT_RightWESInterface.Field[#sa_RightCubby[1]].PLC2WES.ContainerID := "DB_GIN".GIN[#sa_TrackingArray590[(#iUDT_Configuration."590".PEC_Eos.Distance / 10) - 1]].General.Identification.Barcode;
	                                #iqUDT_RightWESInterface.Field[#sa_RightCubby[1]].PLC2WES.SetContainerID := TRUE;
	                            END_IF;

	                        ELSE
	                            IF #iqUDT_RightWESInterface.Field[#sa_RightCubby[1]].PLC2WES.ContainerID <> #cs_MissingBarcodeCode
	                            THEN
	                                #iqUDT_RightWESInterface.Field[#sa_RightCubby[1]].PLC2WES.ContainerID := #cs_MissingBarcodeCode;
	                                #iqUDT_RightWESInterface.Field[#sa_RightCubby[1]].PLC2WES.SetContainerID := TRUE;

	                            END_IF;

	                        END_IF;
	                    END_REGION ;
	                    REGION 580
	                        // second position
	                        //
	                        IF NOT #iqUDT_WorkstationStatus."580".PEC_EoS.PEC
	                            AND #sa_TrackingArray580[(#iUDT_Configuration."580".PEC_Eos.Distance / 10) - 1] > 0
	                        THEN

	                            IF #iqUDT_RightWESInterface.Field[#sa_RightCubby[2]].WES2PLC.SetContainerID THEN

	                                "DB_GIN".GIN[#sa_TrackingArray580[(#iUDT_Configuration."580".PEC_Eos.Distance / 10) - 1]].General.Identification.Barcode := #iqUDT_RightWESInterface.Field[#sa_RightCubby[2]].WES2PLC.ContainerID;
	                                #iqUDT_RightWESInterface.Field[#sa_RightCubby[2]].WES2PLC.SetContainerID := FALSE;

	                            END_IF;

	                            IF #iqUDT_RightWESInterface.Field[#sa_RightCubby[2]].PLC2WES.ContainerID <> "DB_GIN".GIN[#sa_TrackingArray580[(#iUDT_Configuration."580".PEC_Eos.Distance / 10) - 1]].General.Identification.Barcode
	                            THEN

	                                #iqUDT_RightWESInterface.Field[#sa_RightCubby[2]].PLC2WES.ContainerID := "DB_GIN".GIN[#sa_TrackingArray580[(#iUDT_Configuration."580".PEC_Eos.Distance / 10) - 1]].General.Identification.Barcode;
	                                #iqUDT_RightWESInterface.Field[#sa_RightCubby[2]].PLC2WES.SetContainerID := TRUE;
	                            END_IF;

	                        ELSE
	                            IF #iqUDT_RightWESInterface.Field[#sa_RightCubby[2]].PLC2WES.ContainerID <> #cs_MissingBarcodeCode
	                            THEN
	                                #iqUDT_RightWESInterface.Field[#sa_RightCubby[2]].PLC2WES.ContainerID := #cs_MissingBarcodeCode;
	                                #iqUDT_RightWESInterface.Field[#sa_RightCubby[2]].PLC2WES.SetContainerID := TRUE;

	                            END_IF;

	                        END_IF;
	                    END_REGION ;
	                    REGION 570
	                        // third position
	                        //
	                        IF NOT #iqUDT_WorkstationStatus."570".PEC_EoS.PEC
	                            AND #sa_TrackingArray570[(#iUDT_Configuration."570".PEC_Eos.Distance / 10) - 1] > 0
	                        THEN

	                            IF #iqUDT_RightWESInterface.Field[#sa_RightCubby[3]].WES2PLC.SetContainerID THEN

	                                "DB_GIN".GIN[#sa_TrackingArray570[(#iUDT_Configuration."570".PEC_Eos.Distance / 10) - 1]].General.Identification.Barcode := #iqUDT_RightWESInterface.Field[#sa_RightCubby[3]].WES2PLC.ContainerID;
	                                #iqUDT_RightWESInterface.Field[#sa_RightCubby[3]].WES2PLC.SetContainerID := FALSE;

	                            END_IF;

	                            IF #iqUDT_RightWESInterface.Field[#sa_RightCubby[3]].PLC2WES.ContainerID <> "DB_GIN".GIN[#sa_TrackingArray570[(#iUDT_Configuration."570".PEC_Eos.Distance / 10) - 1]].General.Identification.Barcode
	                            THEN

	                                #iqUDT_RightWESInterface.Field[#sa_RightCubby[3]].PLC2WES.ContainerID := "DB_GIN".GIN[#sa_TrackingArray570[(#iUDT_Configuration."570".PEC_Eos.Distance / 10) - 1]].General.Identification.Barcode;
	                                #iqUDT_RightWESInterface.Field[#sa_RightCubby[3]].PLC2WES.SetContainerID := TRUE;
	                            END_IF;

	                        ELSE
	                            IF #iqUDT_RightWESInterface.Field[#sa_RightCubby[3]].PLC2WES.ContainerID <> #cs_MissingBarcodeCode
	                            THEN
	                                #iqUDT_RightWESInterface.Field[#sa_RightCubby[3]].PLC2WES.ContainerID := #cs_MissingBarcodeCode;
	                                #iqUDT_RightWESInterface.Field[#sa_RightCubby[3]].PLC2WES.SetContainerID := TRUE;

	                            END_IF;

	                        END_IF;
	                    END_REGION ;
	                    REGION 560
	                        // fourth position
	                        //
	                        IF NOT #iqUDT_WorkstationStatus."560".PEC_EoS.PEC
	                            AND #sa_TrackingArray560[(#iUDT_Configuration."560".PEC_Eos.Distance / 10) - 1] > 0
	                        THEN

	                            IF #iqUDT_RightWESInterface.Field[#sa_RightCubby[4]].WES2PLC.SetContainerID THEN

	                                "DB_GIN".GIN[#sa_TrackingArray560[(#iUDT_Configuration."560".PEC_Eos.Distance / 10) - 1]].General.Identification.Barcode := #iqUDT_RightWESInterface.Field[#sa_RightCubby[4]].WES2PLC.ContainerID;
	                                #iqUDT_RightWESInterface.Field[#sa_RightCubby[4]].WES2PLC.SetContainerID := FALSE;

	                            END_IF;

	                            IF #iqUDT_RightWESInterface.Field[#sa_RightCubby[4]].PLC2WES.ContainerID <> "DB_GIN".GIN[#sa_TrackingArray560[(#iUDT_Configuration."560".PEC_Eos.Distance / 10) - 1]].General.Identification.Barcode
	                            THEN

	                                #iqUDT_RightWESInterface.Field[#sa_RightCubby[4]].PLC2WES.ContainerID := "DB_GIN".GIN[#sa_TrackingArray560[(#iUDT_Configuration."560".PEC_Eos.Distance / 10) - 1]].General.Identification.Barcode;
	                                #iqUDT_RightWESInterface.Field[#sa_RightCubby[4]].PLC2WES.SetContainerID := TRUE;
	                            END_IF;

	                        ELSE
	                            IF #iqUDT_RightWESInterface.Field[#sa_RightCubby[4]].PLC2WES.ContainerID <> #cs_MissingBarcodeCode
	                            THEN
	                                #iqUDT_RightWESInterface.Field[#sa_RightCubby[4]].PLC2WES.ContainerID := #cs_MissingBarcodeCode;
	                                #iqUDT_RightWESInterface.Field[#sa_RightCubby[4]].PLC2WES.SetContainerID := TRUE;

	                            END_IF;

	                        END_IF;
	                    END_REGION ;
	                    REGION 550
	                        //fifth position
	                        //
	                        IF NOT #iqUDT_WorkstationStatus."550".PEC_EoS.PEC
	                            AND #sa_TrackingArray550[(#iUDT_Configuration."550".PEC_Eos.Distance / 10) - 1] > 0
	                        THEN

	                            IF #iqUDT_RightWESInterface.Field[#sa_RightCubby[5]].WES2PLC.SetContainerID THEN

	                                "DB_GIN".GIN[#sa_TrackingArray550[(#iUDT_Configuration."550".PEC_Eos.Distance / 10) - 1]].General.Identification.Barcode := #iqUDT_RightWESInterface.Field[#sa_RightCubby[5]].WES2PLC.ContainerID;
	                                #iqUDT_RightWESInterface.Field[#sa_RightCubby[5]].WES2PLC.SetContainerID := FALSE;

	                            END_IF;

	                            IF #iqUDT_RightWESInterface.Field[#sa_RightCubby[5]].PLC2WES.ContainerID <> "DB_GIN".GIN[#sa_TrackingArray550[(#iUDT_Configuration."550".PEC_Eos.Distance / 10) - 1]].General.Identification.Barcode
	                            THEN

	                                #iqUDT_RightWESInterface.Field[#sa_RightCubby[5]].PLC2WES.ContainerID := "DB_GIN".GIN[#sa_TrackingArray550[(#iUDT_Configuration."550".PEC_Eos.Distance / 10) - 1]].General.Identification.Barcode;
	                                #iqUDT_RightWESInterface.Field[#sa_RightCubby[5]].PLC2WES.SetContainerID := TRUE;
	                            END_IF;

	                        ELSE
	                            IF #iqUDT_RightWESInterface.Field[#sa_RightCubby[5]].PLC2WES.ContainerID <> #cs_MissingBarcodeCode
	                            THEN
	                                #iqUDT_RightWESInterface.Field[#sa_RightCubby[5]].PLC2WES.ContainerID := #cs_MissingBarcodeCode;
	                                #iqUDT_RightWESInterface.Field[#sa_RightCubby[5]].PLC2WES.SetContainerID := TRUE;

	                            END_IF;

	                        END_IF;
	                    END_REGION ;

	                END_IF;


	            END_REGION

	        END_REGION

	        REGION 6.4 - Function block calls
	            REGION 510

	                REGION Displacement

	                    #sFB_Displacement510(#sUDT_Interface510);

	                END_REGION

	                REGION Conveyor

	                    #sFB_Conveyor510(iUDT_ConveyorConfiguration := #iUDT_Configuration."510".Conveyor,
	                                     idi_PECEoSDistance := 0,
	                                     idi_PECBoSDistance := 0,
	                                     ii_ExternalSpeed := 0,
	                                     ix_SafetyOk := #ix_SafetyOk,
	                                     ix_24vOk := #ix_24vOk,
	                                     ix_400vOk := #ix_400vOk,
	                                     ix_HardwareOk := #iUDT_HardwareOk."510",
	                                     ix_PECEoS := TRUE,
	                                     ix_PECBoS := TRUE,
	                                     ix_ReverseDirection := FALSE,
	                                     ix_ExternalRequestDieBack := FALSE,
	                                     ix_ExternalRequestHold := FALSE,
	                                     ix_ResetEnergySave := FALSE,
	                                     qUDT_HMIStatus => #iqUDT_WorkstationStatus."510".Conveyor,
	                                     qUDT_Status => #iqUDT_WorkstationCommonStatus."510",
	                                     iqUDT_EquipmentControl := #iqUDT_EquipmentControl,
	                                     iqUDT_ConveyorCommand := #iqUDT_WorkstationCommands."510".Conveyor,
	                                     iqUDT_ConveyorInterface := #sUDT_Interface510,
	                                     iqUDT_HandShakeUp := #sUDT_Handshake510A,
	                                     iqUDT_HandShake := #sUDT_Handshake510,
	                                     iqUDT_Statistics := #iqUDT_WorkstationStatistics."510".Conveyor);
	                END_REGION

	                REGION MCO

	                    #sFB_MCOConveyLinxAixController510(iUDT_AixConfig := #iUDT_Configuration."510".MCO_M01,
	                                                       iv_AixInputsModule := #iUDT_MotorInput510,
	                                                       ix_24vOk := #ix_24vOk,
	                                                       ix_SimulationModeActive := "DB_Memory".Simulation,
	                                                       ii_MotorPositionId := 1,
	                                                       qUDT_HMIStatus => #iqUDT_WorkstationStatus."510".MCO_M01,
	                                                       iqv_AixOutputsModule := #iqUDT_MotorOutput510,
	                                                       iqUDT_ConveyorInterface := #sUDT_Interface510,
	                                                       iqUDT_MCOStatistics := #iqUDT_WorkstationStatistics."510".MCO_M01);
	                END_REGION
	            END_REGION

	            REGION 520

	                REGION Displacement

	                    #sFB_Displacement520(#sUDT_Interface520);

	                END_REGION

	                REGION Tracking
	                    #sFB_Tracking520(iUDT_ConveyorCommonConfiguration := #iUDT_Configuration."520".Conveyor.Common,
	                                     iqa_TrackingData := #sa_TrackingArray520,
	                                     iqUDT_ConveyorInterface := #sUDT_Interface520,
	                                     iqUDT_HandshakeUp := #sUDT_Handshake510,
	                                     iqUDT_Handshake := #sUDT_Handshake520);

	                END_REGION


	                REGION EOS

	                    #sFB_PECUpdate520(iUDT_PECUpdateConfiguration := #iUDT_Configuration."520".PEC_Eos,
	                                      iUDT_ConveyorCommonConfiguration := #iUDT_Configuration."520".Conveyor.Common,
	                                      ix_PEC := #iUDT_MotorInput520.AllSensorPortInputs.LeftSensor,
	                                      ix_TeachingMode := FALSE,
	                                      qUDT_Status => #iqUDT_WorkstationStatus."520".PEC_EoS,
	                                      qi_GINwrite => #ti_dummy,
	                                      qx_PECFiltered => #tx_dummy,
	                                      iqUDT_ConveyorInterface := #sUDT_Interface520,
	                                      iqUDT_UnknownGINRange := #iqUDT_UnknownGINRange,
	                                      iqUDT_FifoHeader := "DB_FIFOLostGIN".Header,
	                                      iqUDT_Statistics := #iqUDT_WorkstationStatistics."520".PEC_EoS,
	                                      iqa_TrackingData := #sa_TrackingArray520,
	                                      iqa_FifoData := "DB_FIFOLostGIN".Data);

	                END_REGION

	                REGION Conveyor

	                    #sFB_Conveyor520(iUDT_ConveyorConfiguration := #iUDT_Configuration."520".Conveyor,
	                                     idi_PECEoSDistance := #iUDT_Configuration."520".PEC_Eos.Distance,
	                                     idi_PECBoSDistance := 0,
	                                     ii_ExternalSpeed := 0,
	                                     ix_SafetyOk := #ix_SafetyOk,
	                                     ix_24vOk := #ix_24vOk,
	                                     ix_400vOk := #ix_400vOk,
	                                     ix_HardwareOk := #iUDT_HardwareOk."520",
	                                     ix_PECEoS := #iqUDT_WorkstationStatus."520".PEC_EoS.PEC,
	                                     ix_PECBoS := TRUE,
	                                     ix_ReverseDirection := FALSE,
	                                     ix_ExternalRequestDieBack := FALSE,
	                                     ix_ExternalRequestHold := FALSE,
	                                     ix_ResetEnergySave := FALSE,
	                                     qUDT_HMIStatus => #iqUDT_WorkstationStatus."520".Conveyor,
	                                     qUDT_Status => #iqUDT_WorkstationCommonStatus."520",
	                                     iqUDT_EquipmentControl := #iqUDT_EquipmentControl,
	                                     iqUDT_ConveyorCommand := #iqUDT_WorkstationCommands."520".Conveyor,
	                                     iqUDT_ConveyorInterface := #sUDT_Interface520,
	                                     iqUDT_HandShakeUp := #sUDT_Handshake510,
	                                     iqUDT_HandShake := #sUDT_Handshake520,
	                                     iqUDT_Statistics := #iqUDT_WorkstationStatistics."520".Conveyor);
	                END_REGION

	                REGION MCO

	                    #sFB_MCOConveyLinxAixController520(iUDT_AixConfig := #iUDT_Configuration."520".MCO_M01,
	                                                       iv_AixInputsModule := #iUDT_MotorInput520,
	                                                       ix_24vOk := #ix_24vOk,
	                                                       ix_SimulationModeActive := "DB_Memory".Simulation,
	                                                       ii_MotorPositionId := 1,
	                                                       qUDT_HMIStatus => #iqUDT_WorkstationStatus."520".MCO_M01,
	                                                       iqv_AixOutputsModule := #iqUDT_MotorOutput520,
	                                                       iqUDT_ConveyorInterface := #sUDT_Interface520,
	                                                       iqUDT_MCOStatistics := #iqUDT_WorkstationStatistics."520".MCO_M01);
	                END_REGION
	            END_REGION

	            REGION 521
	                REGION Scanner

	                    #sFB_DataLogicBlade521(iUDT_ScannerInput := #iUDT_ScannerInput521,
	                                           iUDT_ScannerConfiguration := #iUDT_Configuration."521".Scanner,
	                                           ii_GIN := #sa_TrackingArray520[#iUDT_Configuration."521".Scanner.ScannerPosition],
	                                           ix_24vOk := #ix_24vOk,
	                                           ix_HardwareOk := #iUDT_HardwareOk."521",
	                                           ix_SimulationModeActive := "DB_Memory".Simulation,
	                                           qUDT_ScannerOutput => #qUDT_ScannerOutput521,
	                                           qUDT_HMIStatus => #iqUDT_WorkstationStatus."521".Scanner,
	                                           qUDT_CommonStatus => #iqUDT_WorkstationCommonStatus."521",
	                                           iqUDT_Statistics := #iqUDT_WorkstationStatistics."521".Scanner,
	                                           iqUDT_EquipmentControl := #iqUDT_EquipmentControl);



	                END_REGION
	            END_REGION

	            REGION 530

	                REGION Displacement

	                    #sFB_Displacement530(#sUDT_Interface530);

	                END_REGION

	                REGION Tracking

	                    #sFB_Tracking530(iUDT_ConveyorCommonConfiguration := #iUDT_Configuration."530".Conveyor.Common,
	                                     iqa_TrackingData := #sa_TrackingArray530,
	                                     iqUDT_ConveyorInterface := #sUDT_Interface530,
	                                     iqUDT_HandshakeUp := #sUDT_Handshake520,
	                                     iqUDT_Handshake := #sUDT_Handshake530);

	                END_REGION

	                REGION EOS

	                    #sFB_PECUpdate530(iUDT_PECUpdateConfiguration := #iUDT_Configuration."530".PEC_Eos,
	                                      iUDT_ConveyorCommonConfiguration := #iUDT_Configuration."530".Conveyor.Common,
	                                      ix_PEC := #iUDT_MotorInput520.AllSensorPortInputs.RightSensor,
	                                      ix_TeachingMode := FALSE,
	                                      qUDT_Status => #iqUDT_WorkstationStatus."530".PEC_EoS,
	                                      qi_GINwrite => #ti_dummy,
	                                      qx_PECFiltered => #tx_dummy,
	                                      iqUDT_ConveyorInterface := #sUDT_Interface530,
	                                      iqUDT_UnknownGINRange := #iqUDT_UnknownGINRange,
	                                      iqUDT_FifoHeader := "DB_FIFOLostGIN".Header,
	                                      iqUDT_Statistics := #iqUDT_WorkstationStatistics."530".PEC_EoS,
	                                      iqa_TrackingData := #sa_TrackingArray530,
	                                      iqa_FifoData := "DB_FIFOLostGIN".Data);

	                END_REGION

	                REGION Conveyor

	                    #sUDT_Handshake530.RTR := #iqUDT_WorkstationStatus."530".PEC_EoS.PEC OR
	                    (#iqUDT_WorkstationStatus."540".PEC_EoS.PEC AND #sUDT_Interface540.ActualSpeed <> 0);

	                    #sFB_Conveyor530(iUDT_ConveyorConfiguration := #iUDT_Configuration."530".Conveyor,
	                                     idi_PECEoSDistance := #iUDT_Configuration."530".PEC_Eos.Distance,
	                                     idi_PECBoSDistance := 0,
	                                     ii_ExternalSpeed := 0,
	                                     ix_SafetyOk := #ix_SafetyOk,
	                                     ix_24vOk := #ix_24vOk,
	                                     ix_400vOk := #ix_400vOk,
	                                     ix_HardwareOk := #iUDT_HardwareOk."530",
	                                     ix_PECEoS := #iqUDT_WorkstationStatus."530".PEC_EoS.PEC,
	                                     ix_PECBoS := TRUE,
	                                     ix_ReverseDirection := FALSE,
	                                     ix_ExternalRequestDieBack := FALSE,
	                                     ix_ExternalRequestHold := FALSE,
	                                     ix_ResetEnergySave := FALSE,
	                                     qUDT_HMIStatus => #iqUDT_WorkstationStatus."530".Conveyor,
	                                     qUDT_Status => #iqUDT_WorkstationCommonStatus."530",
	                                     iqUDT_EquipmentControl := #iqUDT_EquipmentControl,
	                                     iqUDT_ConveyorCommand := #iqUDT_WorkstationCommands."530".Conveyor,
	                                     iqUDT_ConveyorInterface := #sUDT_Interface530,
	                                     iqUDT_HandShakeUp := #sUDT_Handshake520,
	                                     iqUDT_HandShake := #sUDT_Handshake530,
	                                     iqUDT_Statistics := #iqUDT_WorkstationStatistics."530".Conveyor);
	                END_REGION

	                REGION MCO

	                    #sFB_MCOConveyLinxAixController530(iUDT_AixConfig := #iUDT_Configuration."530".MCO_M01,
	                                                       iv_AixInputsModule := #iUDT_MotorInput520,
	                                                       ix_24vOk := #ix_24vOk,
	                                                       ix_SimulationModeActive := "DB_Memory".Simulation,
	                                                       ii_MotorPositionId := 2,
	                                                       qUDT_HMIStatus => #iqUDT_WorkstationStatus."530".MCO_M01,
	                                                       iqv_AixOutputsModule := #iqUDT_MotorOutput520,
	                                                       iqUDT_ConveyorInterface := #sUDT_Interface530,
	                                                       iqUDT_MCOStatistics := #iqUDT_WorkstationStatistics."530".MCO_M01);
	                END_REGION

	            END_REGION

	            REGION 540

	                REGION Displacement

	                    #sFB_Displacement540(#sUDT_Interface540);

	                END_REGION

	                REGION MCO

	                    #sFB_MCOConveyLinxAixController540(iUDT_AixConfig := #iUDT_Configuration."540".MCO_M01,
	                                                       iv_AixInputsModule := #iUDT_MotorInput540,
	                                                       ii_PositionSetpoint := #iqUDT_RATPositioning540.Lower.EndPosition,
	                                                       ix_24vOk := #ix_24vOk,
	                                                       ix_SimulationModeActive := "DB_Memory".Simulation,
	                                                       ii_MotorPositionId := 1,
	                                                       ix_StartPositioning := #iqUDT_RATPositioning540.Lower.Start,
	                                                       ix_ResetPosition := #iqUDT_RATPositioning540.Lower.ResetPosition,
	                                                       qUDT_HMIStatus => #iqUDT_WorkstationStatus."540".MCO_M01,
	                                                       qx_Positioned => #iqUDT_RATPositioning540.Lower.Done,
	                                                       iqv_AixOutputsModule := #iqUDT_MotorOutput540,
	                                                       iqUDT_ConveyorInterface := #sUDT_Interface540,
	                                                       iqUDT_MCOStatistics := #iqUDT_WorkstationStatistics."540".MCO_M01);
	                END_REGION
	            END_REGION

	            REGION 541

	                REGION Displacement

	                    #sFB_Displacement541(#sUDT_Interface541);

	                END_REGION

	                REGION RAT
	                    #sUDT_Handshake541.RTR := #sx_RightIndexing AND
	                    (#iqUDT_WorkstationStatus."550".PEC_EoS.PEC AND #sUDT_Interface550.ActualSpeed <> 0);

	                    #sFB_RightAngledTransfer541(iUDT_Configuration := #iUDT_Configuration."541".RightAngledTransfer,
	                                                iUDT_LowerConveyorConfiguration := #iUDT_Configuration."540".Conveyor,
	                                                iUDT_UpperConveyorConfiguration := #iUDT_Configuration."541".Conveyor,
	                                                iUDT_PECConfiguration := #iUDT_Configuration."540".PEC_EoS,
	                                                ii_DestinationA := #si_RightDestinationD541,
	                                                ii_DestinationB := 0,
	                                                ii_DestinationC := 0,
	                                                ii_DestinationD := 0,
	                                                ix_HardwareOk := #iUDT_HardwareOk."540",
	                                                ix_400vOk := #ix_400vOk,
	                                                ix_24vOk := #ix_24vOk,
	                                                ix_SafetyOk := #ix_SafetyOk,
	                                                ix_AirPressureOk := #ix_AirPressureOk,
	                                                ix_SectionIsDown := #ix_SectionIsDown541,
	                                                ix_SectionIsUp := #ix_SectionIsUp541,
	                                                ix_ConveyorAAuto := #iqUDT_WorkstationCommonStatus."530".AutoON,
	                                                ix_ConveyorBAuto := false,
	                                                ix_ConveyorCAuto := false,
	                                                ix_ConveyorDAuto := false,
	                                                ix_PEC := #iUDT_MotorInput540.AllSensorPortInputs.LeftSensor,
	                                                ix_ExternalReceiveRequestA := NOT #iqUDT_WorkstationStatus."530".PEC_EoS.PEC,
	                                                ix_ExternalReceiveRequestB := FALSE,
	                                                ix_ExternalReceiveRequestC := FALSE,
	                                                ix_ExternalReceiveRequestD := FALSE,
	                                                ix_PECInfeedA := #iqUDT_WorkstationStatus."530".PEC_EoS.PEC,
	                                                qUDT_HMIRATStatus => #iqUDT_WorkstationStatus."541".RightAngledTransfer,
	                                                qUDT_HMIConveyorStatus => #iqUDT_WorkstationStatus."540".Conveyor,
	                                                qUDT_HMIPECStatus => #iqUDT_WorkstationStatus."540".PEC_EoS,
	                                                qUDT_RATStatus => #iqUDT_WorkstationCommonStatus."541",
	                                                qUDT_ConveyorStatus => #iqUDT_WorkstationCommonStatus."540",
	                                                qx_PopupControl => #qx_PopupControl541,
	                                                qx_ExternalSendRequestA => #tx_dummy,
	                                                qx_ExternalSendRequestB => #tx_dummy,
	                                                qx_ExternalSendRequestC => #tx_dummy,
	                                                qx_ExternalSendRequestD => #tx_dummy,
	                                                iqUDT_EquipmentControl := #iqUDT_EquipmentControl,
	                                                iqUDT_RATCommand := #iqUDT_WorkstationCommands."541".RightAngledTransfer,
	                                                iqUDT_ConveyorCommand := #iqUDT_WorkstationCommands."540".Conveyor,
	                                                iqUDT_RATStatistics := #iqUDT_WorkstationStatistics."541".RightAngledTransfer,
	                                                iqUDT_ConveyorStatistics := #iqUDT_WorkstationStatistics."540".Conveyor,
	                                                iqUDT_PECStatistics := #iqUDT_WorkstationStatistics."540".PEC_EoS,
	                                                iqUDT_HandShakeConveyorA := #sUDT_Handshake530,
	                                                iqUDT_HandShakeConveyorB := #tUDT_DummyConveyorHandshake,
	                                                iqUDT_HandShakeConveyorC := #tUDT_DummyConveyorHandshake,
	                                                iqUDT_HandShakeConveyorD := #sUDT_Handshake541,
	                                                iqUDT_LowerConveyorInterface := #sUDT_Interface540,
	                                                iqUDT_UpperConveyorInterface := #sUDT_Interface541,
	                                                iqUDT_RATPositioning := #iqUDT_RATPositioning540,
	                                                iqUDT_BladeStopEoSInterface := #tUDT_DummyBladeStop,
	                                                iqUDT_BladeStopBoSInterface := #tUDT_DummyBladeStop);

	                END_REGION

	                REGION MCO

	                    #sFB_MCOConveyLinxAixController541(iUDT_AixConfig := #iUDT_Configuration."541".MCO_M01,
	                                                       iv_AixInputsModule := #iUDT_MotorInput540,
	                                                       ix_24vOk := #ix_24vOk,
	                                                       ix_SimulationModeActive := "DB_Memory".Simulation,
	                                                       ii_MotorPositionId := 2,
	                                                       qUDT_HMIStatus => #iqUDT_WorkstationStatus."541".MCO_M01,
	                                                       iqv_AixOutputsModule := #iqUDT_MotorOutput540,
	                                                       iqUDT_ConveyorInterface := #sUDT_Interface541,
	                                                       iqUDT_MCOStatistics := #iqUDT_WorkstationStatistics."541".MCO_M01);
	                END_REGION

	            END_REGION

	            REGION 550

	                REGION Displacement

	                    #sFB_Displacement550(#sUDT_Interface550);

	                END_REGION

	                REGION Tracking

	                    #sFB_Tracking550(iUDT_ConveyorCommonConfiguration := #iUDT_Configuration."550".Conveyor.Common,
	                                     iqa_TrackingData := #sa_TrackingArray550,
	                                     iqUDT_ConveyorInterface := #sUDT_Interface550,
	                                     iqUDT_HandshakeUp := #sUDT_Handshake541,
	                                     iqUDT_Handshake := #sUDT_Handshake550);
	                END_REGION

	                REGION EOS

	                    #sFB_PECUpdate550(iUDT_PECUpdateConfiguration := #iUDT_Configuration."550".PEC_Eos,
	                                      iUDT_ConveyorCommonConfiguration := #iUDT_Configuration."550".Conveyor.Common,
	                                      ix_PEC := NOT #iUDT_MotorInput550.AllSensorPortInputs.LeftSensor,
	                                      ix_TeachingMode := FALSE,
	                                      qUDT_Status => #iqUDT_WorkstationStatus."550".PEC_EoS,
	                                      qi_GINwrite => #ti_dummy,
	                                      qx_PECFiltered => #tx_dummy,
	                                      iqa_TrackingData := #sa_TrackingArray550,
	                                      iqUDT_ConveyorInterface := #sUDT_Interface550,
	                                      iqUDT_UnknownGINRange := #iqUDT_UnknownGINRange,
	                                      iqUDT_FifoHeader := "DB_FIFOLostGIN".Header,
	                                      iqa_FifoData := "DB_FIFOLostGIN".Data,
	                                      iqUDT_Statistics := #iqUDT_WorkstationStatistics."550".PEC_EoS);

	                END_REGION

	                REGION Conveyor

	                    #sUDT_Handshake550.RTR := #sx_RightIndexing AND
	                    ((#iqUDT_WorkstationStatus."560".PEC_EoS.PEC AND #sUDT_Interface560.ActualSpeed <> 0) OR #iqUDT_WorkstationStatus."550".PEC_EoS.PEC);

	                    #sFB_Conveyor550(iUDT_ConveyorConfiguration := #iUDT_Configuration."550".Conveyor,
	                                     idi_PECEoSDistance := #iUDT_Configuration."550".PEC_Eos.Distance,
	                                     idi_PECBoSDistance := 0,
	                                     ii_ExternalSpeed := 0,
	                                     ix_SafetyOk := #ix_SafetyOk,
	                                     ix_24vOk := #ix_24vOk,
	                                     ix_400vOk := #ix_400vOk,
	                                     ix_HardwareOk := #iUDT_HardwareOk."550",
	                                     ix_PECEoS := #iqUDT_WorkstationStatus."550".PEC_EoS.PEC,
	                                     ix_PECBoS := TRUE,
	                                     ix_ReverseDirection := FALSE,
	                                     ix_ExternalRequestDieBack := FALSE,
	                                     ix_ExternalRequestHold := #sx_RightExternalRequestHold550,
	                                     ix_ResetEnergySave := FALSE,
	                                     qUDT_HMIStatus => #iqUDT_WorkstationStatus."550".Conveyor,
	                                     qUDT_Status => #iqUDT_WorkstationCommonStatus."550",
	                                     iqUDT_EquipmentControl := #iqUDT_EquipmentControl,
	                                     iqUDT_ConveyorCommand := #iqUDT_WorkstationCommands."550".Conveyor,
	                                     iqUDT_ConveyorInterface := #sUDT_Interface550,
	                                     iqUDT_HandShakeUp := #sUDT_Handshake541,
	                                     iqUDT_HandShake := #sUDT_Handshake550,
	                                     iqUDT_Statistics := #iqUDT_WorkstationStatistics."550".Conveyor);
	                END_REGION

	                REGION MCO

	                    #sFB_MCOConveyLinxAixController550(iUDT_AixConfig := #iUDT_Configuration."550".MCO_M01,
	                                                       iv_AixInputsModule := #iUDT_MotorInput550,
	                                                       ix_24vOk := #ix_24vOk,
	                                                       ix_SimulationModeActive := "DB_Memory".Simulation,
	                                                       ii_MotorPositionId := 1,
	                                                       qUDT_HMIStatus => #iqUDT_WorkstationStatus."550".MCO_M01,
	                                                       iqv_AixOutputsModule := #iqUDT_MotorOutput550,
	                                                       iqUDT_ConveyorInterface := #sUDT_Interface550,
	                                                       iqUDT_MCOStatistics := #iqUDT_WorkstationStatistics."550".MCO_M01);
	                END_REGION
	            END_REGION

	            REGION 560

	                REGION Displacement

	                    #sFB_Displacement560(#sUDT_Interface560);

	                END_REGION

	                REGION Tracking

	                    #sFB_Tracking560(iUDT_ConveyorCommonConfiguration := #iUDT_Configuration."560".Conveyor.Common,
	                                     iqa_TrackingData := #sa_TrackingArray560,
	                                     iqUDT_ConveyorInterface := #sUDT_Interface560,
	                                     iqUDT_HandshakeUp := #sUDT_Handshake550,
	                                     iqUDT_Handshake := #sUDT_Handshake560);
	                END_REGION

	                REGION EOS

	                    #sFB_PECUpdate560(iUDT_PECUpdateConfiguration := #iUDT_Configuration."560".PEC_Eos,
	                                      iUDT_ConveyorCommonConfiguration := #iUDT_Configuration."560".Conveyor.Common,
	                                      ix_PEC := NOT #iUDT_MotorInput550.AllSensorPortInputs.RightSensor,
	                                      ix_TeachingMode := FALSE,
	                                      qUDT_Status => #iqUDT_WorkstationStatus."560".PEC_EoS,
	                                      qi_GINwrite => #ti_dummy,
	                                      qx_PECFiltered => #tx_dummy,
	                                      iqa_TrackingData := #sa_TrackingArray560,
	                                      iqUDT_ConveyorInterface := #sUDT_Interface560,
	                                      iqUDT_UnknownGINRange := #iqUDT_UnknownGINRange,
	                                      iqUDT_FifoHeader := "DB_FIFOLostGIN".Header,
	                                      iqa_FifoData := "DB_FIFOLostGIN".Data,
	                                      iqUDT_Statistics := #iqUDT_WorkstationStatistics."560".PEC_EoS);

	                END_REGION

	                REGION Conveyor

	                    #sUDT_Handshake560.RTR := #sx_RightIndexing AND
	                    ((#iqUDT_WorkstationStatus."570".PEC_EoS.PEC AND #sUDT_Interface570.ActualSpeed <> 0) OR #iqUDT_WorkstationStatus."560".PEC_EoS.PEC);

	                    #sFB_Conveyor560(iUDT_ConveyorConfiguration := #iUDT_Configuration."560".Conveyor,
	                                     idi_PECEoSDistance := #iUDT_Configuration."560".PEC_Eos.Distance,
	                                     idi_PECBoSDistance := 0,
	                                     ii_ExternalSpeed := 0,
	                                     ix_SafetyOk := #ix_SafetyOk,
	                                     ix_24vOk := #ix_24vOk,
	                                     ix_400vOk := #ix_400vOk,
	                                     ix_HardwareOk := #iUDT_HardwareOk."560",
	                                     ix_PECEoS := #iqUDT_WorkstationStatus."560".PEC_EoS.PEC,
	                                     ix_PECBoS := TRUE,
	                                     ix_ReverseDirection := FALSE,
	                                     ix_ExternalRequestDieBack := FALSE,
	                                     ix_ExternalRequestHold := #sx_RightExternalRequestHold560,
	                                     ix_ResetEnergySave := FALSE,
	                                     qUDT_HMIStatus => #iqUDT_WorkstationStatus."560".Conveyor,
	                                     qUDT_Status => #iqUDT_WorkstationCommonStatus."560",
	                                     iqUDT_EquipmentControl := #iqUDT_EquipmentControl,
	                                     iqUDT_ConveyorCommand := #iqUDT_WorkstationCommands."560".Conveyor,
	                                     iqUDT_ConveyorInterface := #sUDT_Interface560,
	                                     iqUDT_HandShakeUp := #sUDT_Handshake550,
	                                     iqUDT_HandShake := #sUDT_Handshake560,
	                                     iqUDT_Statistics := #iqUDT_WorkstationStatistics."560".Conveyor);
	                END_REGION

	                REGION MCO

	                    #sFB_MCOConveyLinxAixController560(iUDT_AixConfig := #iUDT_Configuration."560".MCO_M01,
	                                                       iv_AixInputsModule := #iUDT_MotorInput550,
	                                                       ix_24vOk := #ix_24vOk,
	                                                       ix_SimulationModeActive := "DB_Memory".Simulation,
	                                                       ii_MotorPositionId := 2,
	                                                       qUDT_HMIStatus => #iqUDT_WorkstationStatus."560".MCO_M01,
	                                                       iqv_AixOutputsModule := #iqUDT_MotorOutput550,
	                                                       iqUDT_ConveyorInterface := #sUDT_Interface560,
	                                                       iqUDT_MCOStatistics := #iqUDT_WorkstationStatistics."560".MCO_M01);
	                END_REGION

	            END_REGION

	            REGION 570

	                REGION Displacement

	                    #sFB_Displacement570(#sUDT_Interface570);

	                END_REGION

	                REGION Tracking

	                    #sFB_Tracking570(iUDT_ConveyorCommonConfiguration := #iUDT_Configuration."570".Conveyor.Common,
	                                     iqa_TrackingData := #sa_TrackingArray570,
	                                     iqUDT_ConveyorInterface := #sUDT_Interface570,
	                                     iqUDT_HandshakeUp := #sUDT_Handshake560,
	                                     iqUDT_Handshake := #sUDT_Handshake570);
	                END_REGION

	                REGION EOS

	                    #sFB_PECUpdate570(iUDT_PECUpdateConfiguration := #iUDT_Configuration."570".PEC_Eos,
	                                      iUDT_ConveyorCommonConfiguration := #iUDT_Configuration."570".Conveyor.Common,
	                                      ix_PEC := NOT #iUDT_MotorInput570.AllSensorPortInputs.LeftSensor,
	                                      ix_TeachingMode := FALSE,
	                                      qUDT_Status => #iqUDT_WorkstationStatus."570".PEC_EoS,
	                                      qi_GINwrite => #ti_dummy,
	                                      qx_PECFiltered => #tx_dummy,
	                                      iqa_TrackingData := #sa_TrackingArray570,
	                                      iqUDT_ConveyorInterface := #sUDT_Interface570,
	                                      iqUDT_UnknownGINRange := #iqUDT_UnknownGINRange,
	                                      iqUDT_FifoHeader := "DB_FIFOLostGIN".Header,
	                                      iqa_FifoData := "DB_FIFOLostGIN".Data,
	                                      iqUDT_Statistics := #iqUDT_WorkstationStatistics."570".PEC_EoS);

	                END_REGION

	                REGION Conveyor

	                    #sUDT_Handshake570.RTR := #sx_RightIndexing AND
	                    ((#iqUDT_WorkstationStatus."580".PEC_EoS.PEC AND #sUDT_Interface580.ActualSpeed <> 0) OR #iqUDT_WorkstationStatus."570".PEC_EoS.PEC);

